FUNCTION_BLOCK LightMode (* Composite Function Block Type *)
  (* Standard: 61499-2 *)
  (* Version 0.0, 2015-05-20, 4DIAC-IDE, 4DIAC-Consortium *)
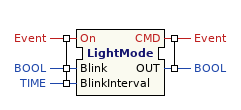
  EVENT_INPUT
    On WITH BlinkInterval, Blink; (* Initialization Request *)
  END_EVENT
  EVENT_OUTPUT
    CMD WITH OUT; (* Initialization Confirm *)
  END_EVENT
  VAR_INPUT
    Blink : BOOL;
    BlinkInterval : TIME; (* Input event qualifier *)
  END_VAR
  VAR_OUTPUT
    OUT : BOOL; (* Output event qualifier *)
  END_VAR
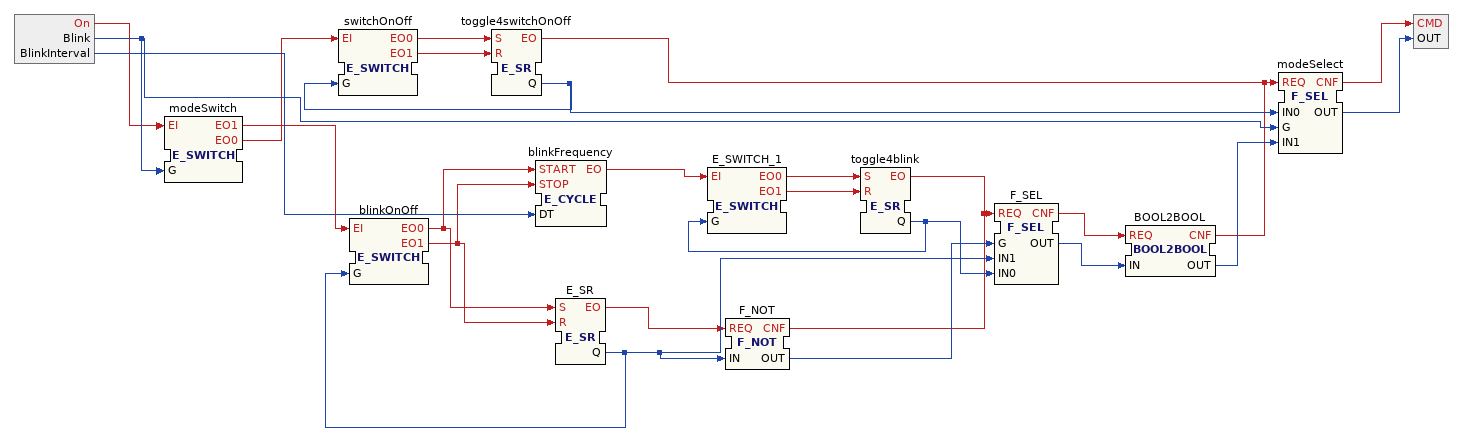
  FBS
    blinkOnOff : E_SWITCH;
    blinkFrequency : E_CYCLE;
    E_SR : E_SR;
    E_SWITCH_1 : E_SWITCH;
    F_NOT : F_NOT;
    toggle4blink : E_SR;
    F_SEL : F_SEL;
    modeSwitch : E_SWITCH;
    switchOnOff : E_SWITCH;
    toggle4switchOnOff : E_SR;
    BOOL2BOOL : BOOL2BOOL;
    modeSelect : F_SEL;
  END_FBS
  EVENT_CONNECTIONS
    blinkOnOff.EO0 TO blinkFrequency.START;
    blinkOnOff.EO0 TO E_SR.S;
    blinkOnOff.EO1 TO blinkFrequency.STOP;
    blinkOnOff.EO1 TO E_SR.R;
    E_SR.EO TO F_NOT.REQ;
    F_NOT.CNF TO F_SEL.REQ;
    toggle4blink.EO TO F_SEL.REQ;
    E_SWITCH_1.EO0 TO toggle4blink.S;
    E_SWITCH_1.EO1 TO toggle4blink.R;
    blinkFrequency.EO TO E_SWITCH_1.EI;
    On TO modeSwitch.EI;
    modeSwitch.EO1 TO blinkOnOff.EI;
    switchOnOff.EO0 TO toggle4switchOnOff.S;
    switchOnOff.EO1 TO toggle4switchOnOff.R;
    modeSwitch.EO0 TO switchOnOff.EI;
    F_SEL.CNF TO BOOL2BOOL.REQ;
    toggle4switchOnOff.EO TO modeSelect.REQ;
    BOOL2BOOL.CNF TO modeSelect.REQ;
    modeSelect.CNF TO CMD;
  END_CONNECTIONS
  DATA_CONNECTIONS
    E_SR.Q TO blinkOnOff.G;
    E_SR.Q TO F_NOT.IN;
    F_NOT.OUT TO F_SEL.G;
    E_SR.Q TO F_SEL.IN1;
    toggle4blink.Q TO F_SEL.IN0;
    toggle4blink.Q TO E_SWITCH_1.G;
    BlinkInterval TO blinkFrequency.DT;
    Blink TO modeSwitch.G;
    toggle4switchOnOff.Q TO switchOnOff.G;
    F_SEL.OUT TO BOOL2BOOL.IN;
    toggle4switchOnOff.Q TO modeSelect.IN0;
    Blink TO modeSelect.G;
    BOOL2BOOL.OUT TO modeSelect.IN1;
    modeSelect.OUT TO OUT;
  END_CONNECTIONS
END_FUNCTION_BLOCK
